FUNCTION_BLOCK FB_TCMLevelEPTUpdate
VAR_INPUT
	iLevel:INT := 0;
END_VAR
VAR_OUTPUT
END_VAR
VAR
	bBlocked 			: BOOL := FALSE;
	bLevelBlocked 		: BOOL := FALSE;
	bEptBlocked 		: BOOL := FALSE;
	bEptBusy 			: BOOL := FALSE;
	bEptIdle 			: BOOL := FALSE;
	stMLVIO				: ST_TCMultiLevel_VIO;
	i					: INT;
END_VAR

//IF iPOC_ML_Selection = 1 AND FALSE THEN
//	bEptBlocked := 	arrTCShuttlePOC[iLevel].stGblParam.iProcessState = E_ProcessState.eALPAUSED OR
//					(*arrTCLevelState[iLevel] = E_State.eDisabled; *) 
//					(TC_ModuleState[iLevel].Tester = E_State.eDisabled OR
//					TC_ModuleState[iLevel].TCSite[1].TCU = E_State.eDisabled OR
//					TC_ModuleState[iLevel].TCSite[1].TIERII = E_State.eDisabled);
//	
//	bEptBusy 	:= 	arrTCShuttlePOC[iLevel].stGblParam.iProcessState = E_ProcessState.eLOADG;
//	bEptIdle 	:= 	arrTCShuttlePOC[iLevel].stGblParam.iProcessState = E_ProcessState.ePAUSE OR
//					arrTCShuttlePOC[iLevel].stGblParam.iProcessState = E_ProcessState.eAWAITGCMD;	
//ELSE
	stMLVIO:=arrTCMultiLevel[iLevel].fbTCMultiLevelSeq.P_stTCMultiLevelVIO;
	
	bEptBlocked := 	(arrTCMultiLevel[iLevel].stGblParam.iProcessState = E_ProcessState.eALPAUSED)	OR	//All alarms besides TIIAlarm block the EPT, Door Recovery executing
					(arrTCMultiLevel[iLevel].stGblParam.iProcessState = E_ProcessState.eUNKNOWN)	OR
					(arrTCMultiLevel[iLevel].stGblParam.bInitialise)								OR //initialization
					(arrTCMultiLevel[iLevel].stGblParam.bDoorRecovery)								OR //Door recovery
					(TC_ModuleState[iLevel].Tester = E_State.eDisabled) 							OR	//tester Modules disabled
					(TC_ModuleState[iLevel].TCSite[1].TCU = E_State.eDisabled) 						OR	//tcu Modules disabled
					 //(TC_ModuleState[iLevel].TCSite[1].TIERII = E_State.eDisabled)				OR	//tier 2 Modules disabled
					(stMLVIO.isSysError) 															OR	//System Facilities OR Column Alarms
					(stMLVIO.TIIAlarmEPT)															OR	//Some TIIAlarms block the EPT
					(NOT stMLVIO.ipTCCellDoorClosed);
				
	bEptBusy 	:= 	(arrTCMultiLevel[iLevel].stGblParam.iProcessState = E_ProcessState.eLOADG)											OR	//executing tasks
					(stMLVIO.ipAPPresentSensor AND (NOT stMLVIO.ipHandlerSafeToEnterHwr OR NOT stMLVIO.ipHandlerSafeToEnterPLC))		OR	//actuate pan actuated with ap present
					(stMLVIO.ipTCDrawerCylUpRS OR stMLVIO.ipTCDrawerCylExtendRS);															//tc drawer up/ out position
	
	bEptIdle 	:= 	arrTCMultiLevel[iLevel].stGblParam.iProcessState = E_ProcessState.ePAUSE OR	
					arrTCMultiLevel[iLevel].stGblParam.iProcessState = E_ProcessState.eAWAITGCMD;	
//END_IF	
	 
IF bEptBlocked THEN 
	//arrTCMLevelEpt[iLevel]:= E_EPT.eBlocked;
	TC_EPT[iLevel].TCSite[1].TCU:=E_EPT.eBlocked;
ELSIF bEptBusy THEN 
	//arrTCMLevelEpt[iLevel]:= E_EPT.eBusy; 
	TC_EPT[iLevel].TCSite[1].TCU:=E_EPT.eBusy;  
ELSIF bEptIdle THEN 
	//arrTCMLevelEpt[iLevel]:= E_EPT.eIdle;   
	TC_EPT[iLevel].TCSite[1].TCU:=E_EPT.eIdle;
END_IF

END_FUNCTION_BLOCK

(* stored: Version 1.1.0.1, ProductVersion 3.1.4022.18
   POU FB_TCMLevelEPTUpdate: Id {a1de3507-2555-4608-93bd-333a14b1f7fe}, SpecialFunc None *)
